// TIA Portal V18 export
TYPE "MEStoPLC_SubCheckIn"
// stored: IsFailsafeCompliant false
   STRUCT
      "M-SubPartDone" : Bool;   // P-ReqSubPart上升沿触发置位，下降沿触发复位
      "M-SubPartOK" : Bool;   // 子零件可加工标志位，PLC收到此信号后可开始加工，P-ReqSubPart下降沿由MES复位此信号
      "M-SubPartNG" : Bool;   // 子零件不可加工标志位，PLC收到此信号后需要重新扫子零件码，P-ReqSubPart下降沿MES复位此信号
      "M-SubPartErrorCode" : Int;   // 【预留】“M-SubPartErrorMsg”失效的时候启用
      "M-SubPartErrorMsg" : String[98];   // P-SubPartReq请求Mes标志位收到后，如果Mes对请求的数据校验有异常，写入相应中文字符串，M-SubPartDone信号超时后将中文字符串显示到HMI
      Reserve : Array[1..196] of Byte;   // SubPartReq子零件绑定交互预留
   END_STRUCT;
END_TYPE
